PROGRAM P_UpdateHmi
VAR_IN_OUT
	Data		: ST_DATA;
END_VAR

Communication.ToHmi.Data	:= Data;

END_PROGRAM

(* stored: Version 1.1.0.1, ProductVersion 3.1.4022.11
   POU P_UpdateHmi: Id {309727f5-7b51-4980-a3c1-d7ca648e43da}, SpecialFunc None *)
